PROGRAM MAIN
VAR
END_VAR

LADDER1();

END_PROGRAM

(* stored: Version 1.1.0.1, ProductVersion 3.1.4018.5
   POU MAIN: Id {55160f5e-0fed-4d94-813d-488b4a3d7b0c}, SpecialFunc None *)
